// TIA Portal V19 export
FUNCTION "MODE SELECTION" : Void   // FC1, LAD
{ S7_Optimized_Access := 'TRUE' }
// stored: SetENOAutomatically false
   VAR_TEMP   // added for the SCL form of the ladder/FBD networks
      _w1 : Bool;
   END_VAR
BEGIN

REGION Network 1: STANDBY///////////////////////////////////// MGF ////////////////////////////////////////
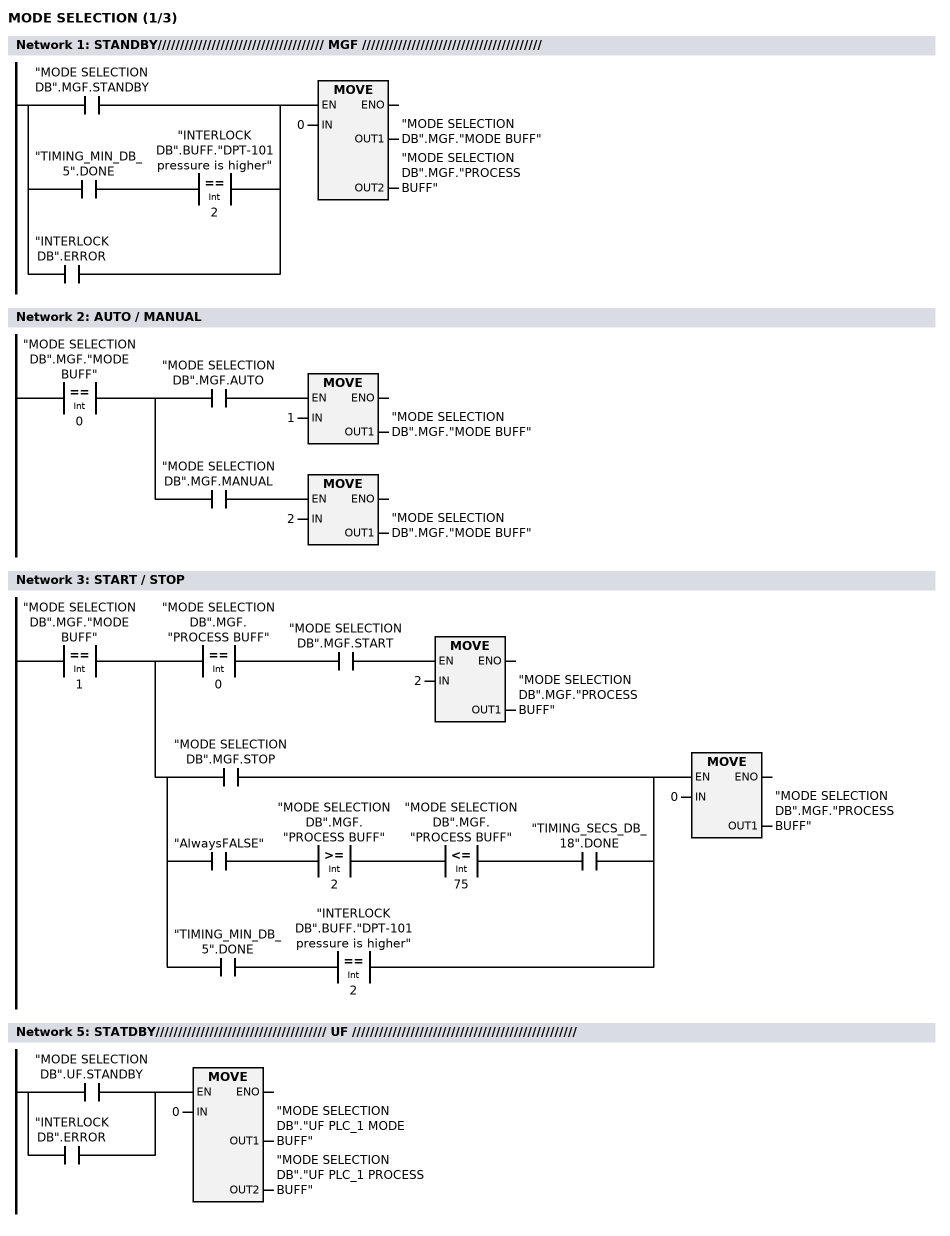
   RUNG wire#powerrail
      Contact( "MODE SELECTION DB".MGF.STANDBY )
      wire#w1
      Move(in := 0, out1 => "MODE SELECTION DB".MGF."MODE BUFF", out2 => "MODE SELECTION DB".MGF."PROCESS BUFF")
   END_RUNG
   RUNG wire#powerrail
      Contact( "TIMING_MIN_DB_5".DONE )
      { S7_Templates := "SrcType := Int" } EQ_Contact(in1 := "INTERLOCK DB".BUFF."DPT-101 pressure is higher", in2 := 2)
   END_RUNG wire#w1
   RUNG wire#powerrail
      Contact( "INTERLOCK DB".ERROR )
   END_RUNG wire#w1
   // the same network as SCL:
   IF "MODE SELECTION DB".MGF.STANDBY OR ("TIMING_MIN_DB_5".DONE AND ("INTERLOCK DB".BUFF."DPT-101 pressure is higher" = 2)) OR "INTERLOCK DB".ERROR THEN
       "MODE SELECTION DB".MGF."MODE BUFF" := 0;
       "MODE SELECTION DB".MGF."PROCESS BUFF" := 0;
   END_IF;
END_REGION

REGION Network 2: AUTO / MANUAL
   RUNG wire#powerrail
      { S7_Templates := "SrcType := Int" } EQ_Contact(in1 := "MODE SELECTION DB".MGF."MODE BUFF", in2 := 0)
      wire#w1
      Contact( "MODE SELECTION DB".MGF.AUTO )
      Move(in := 1, out1 => "MODE SELECTION DB".MGF."MODE BUFF")
   END_RUNG
   RUNG wire#w1
      Contact( "MODE SELECTION DB".MGF.MANUAL )
      Move(in := 2, out1 => "MODE SELECTION DB".MGF."MODE BUFF")
   END_RUNG
   // the same network as SCL:
   #_w1 := "MODE SELECTION DB".MGF."MODE BUFF" = 0;
   IF #_w1 AND "MODE SELECTION DB".MGF.AUTO THEN "MODE SELECTION DB".MGF."MODE BUFF" := 1; END_IF;
   IF #_w1 AND "MODE SELECTION DB".MGF.MANUAL THEN "MODE SELECTION DB".MGF."MODE BUFF" := 2; END_IF;
END_REGION

REGION Network 3: START / STOP
   RUNG wire#powerrail
      { S7_Templates := "SrcType := Int" } EQ_Contact(in1 := "MODE SELECTION DB".MGF."MODE BUFF", in2 := 1)
      wire#w1
      { S7_Templates := "SrcType := Int" } EQ_Contact(in1 := "MODE SELECTION DB".MGF."PROCESS BUFF", in2 := 0)
      Contact( "MODE SELECTION DB".MGF.START )
      Move(in := 2, out1 => "MODE SELECTION DB".MGF."PROCESS BUFF")
   END_RUNG
   RUNG wire#w1
      Contact( "MODE SELECTION DB".MGF.STOP )
      wire#w2
      Move(in := 0, out1 => "MODE SELECTION DB".MGF."PROCESS BUFF")
   END_RUNG
   RUNG wire#w1
      Contact( "AlwaysFALSE" )
      { S7_Templates := "SrcType := Int" } GE_Contact(in1 := "MODE SELECTION DB".MGF."PROCESS BUFF", in2 := 2)
      { S7_Templates := "SrcType := Int" } LE_Contact(in1 := "MODE SELECTION DB".MGF."PROCESS BUFF", in2 := 75)
      Contact( "TIMING_SECS_DB_18".DONE )
   END_RUNG wire#w2
   RUNG wire#w1
      Contact( "TIMING_MIN_DB_5".DONE )
      { S7_Templates := "SrcType := Int" } EQ_Contact(in1 := "INTERLOCK DB".BUFF."DPT-101 pressure is higher", in2 := 2)
   END_RUNG wire#w2
   // the same network as SCL:
   #_w1 := "MODE SELECTION DB".MGF."MODE BUFF" = 1;
   IF #_w1 AND ("MODE SELECTION DB".MGF."PROCESS BUFF" = 0) AND "MODE SELECTION DB".MGF.START THEN
       "MODE SELECTION DB".MGF."PROCESS BUFF" := 2;
   END_IF;
   IF #_w1 AND ("MODE SELECTION DB".MGF.STOP OR ("AlwaysFALSE" AND ("MODE SELECTION DB".MGF."PROCESS BUFF" >= 2) AND ("MODE SELECTION DB".MGF."PROCESS BUFF" <= 75) AND "TIMING_SECS_DB_18".DONE) OR ("TIMING_MIN_DB_5".DONE AND ("INTERLOCK DB".BUFF."DPT-101 pressure is higher" = 2))) THEN
       "MODE SELECTION DB".MGF."PROCESS BUFF" := 0;
   END_IF;
END_REGION

REGION Network 5: STATDBY////////////////////////////////////// UF //////////////////////////////////////////////////
   RUNG wire#powerrail
      Contact( "MODE SELECTION DB".UF.STANDBY )
      wire#w1
      Move(in := 0, out1 => "MODE SELECTION DB"."UF PLC_1 MODE BUFF", out2 => "MODE SELECTION DB"."UF PLC_1 PROCESS BUFF")
   END_RUNG
   RUNG wire#powerrail
      Contact( "INTERLOCK DB".ERROR )
   END_RUNG wire#w1
   // the same network as SCL:
   IF "MODE SELECTION DB".UF.STANDBY OR "INTERLOCK DB".ERROR THEN
       "MODE SELECTION DB"."UF PLC_1 MODE BUFF" := 0;
       "MODE SELECTION DB"."UF PLC_1 PROCESS BUFF" := 0;
   END_IF;
END_REGION

REGION Network 6: AUTO / MANUAL
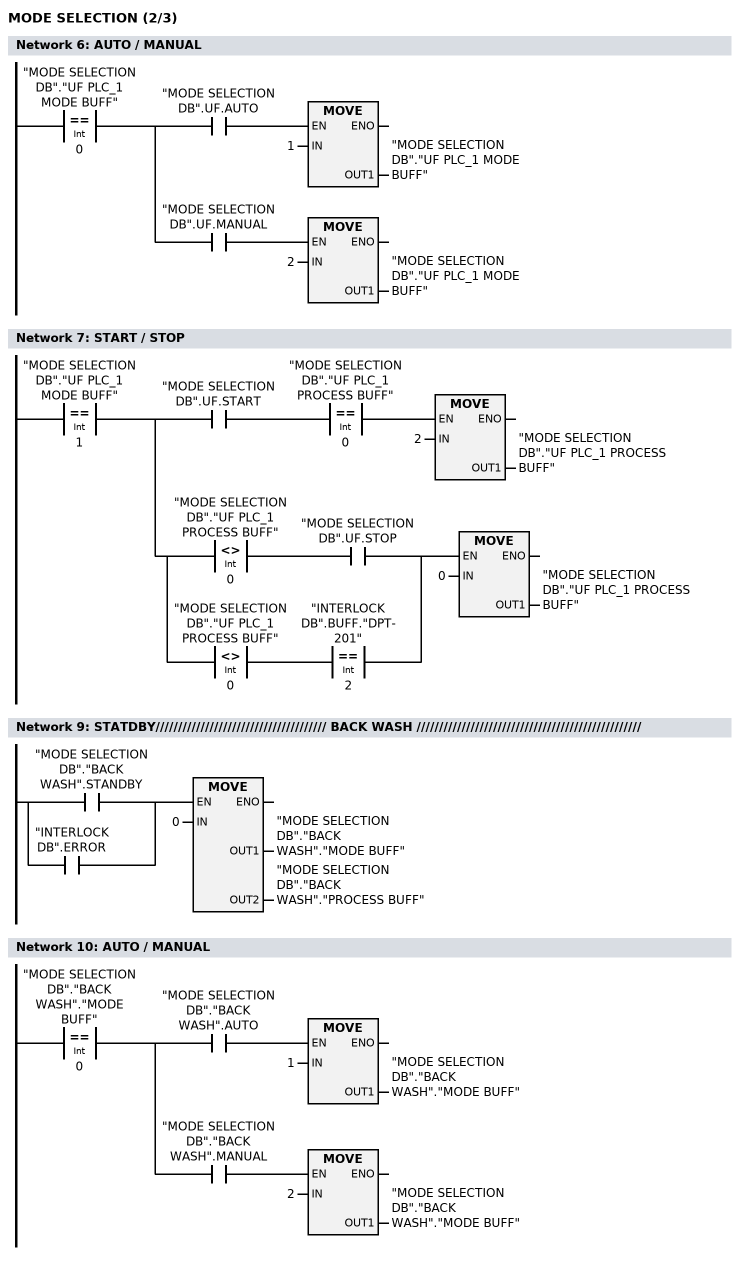
   RUNG wire#powerrail
      { S7_Templates := "SrcType := Int" } EQ_Contact(in1 := "MODE SELECTION DB"."UF PLC_1 MODE BUFF", in2 := 0)
      wire#w1
      Contact( "MODE SELECTION DB".UF.AUTO )
      Move(in := 1, out1 => "MODE SELECTION DB"."UF PLC_1 MODE BUFF")
   END_RUNG
   RUNG wire#w1
      Contact( "MODE SELECTION DB".UF.MANUAL )
      Move(in := 2, out1 => "MODE SELECTION DB"."UF PLC_1 MODE BUFF")
   END_RUNG
   // the same network as SCL:
   #_w1 := "MODE SELECTION DB"."UF PLC_1 MODE BUFF" = 0;
   IF #_w1 AND "MODE SELECTION DB".UF.AUTO THEN "MODE SELECTION DB"."UF PLC_1 MODE BUFF" := 1; END_IF;
   IF #_w1 AND "MODE SELECTION DB".UF.MANUAL THEN "MODE SELECTION DB"."UF PLC_1 MODE BUFF" := 2; END_IF;
END_REGION

REGION Network 7: START / STOP
   RUNG wire#powerrail
      { S7_Templates := "SrcType := Int" } EQ_Contact(in1 := "MODE SELECTION DB"."UF PLC_1 MODE BUFF", in2 := 1)
      wire#w1
      Contact( "MODE SELECTION DB".UF.START )
      { S7_Templates := "SrcType := Int" } EQ_Contact(in1 := "MODE SELECTION DB"."UF PLC_1 PROCESS BUFF", in2 := 0)
      Move(in := 2, out1 => "MODE SELECTION DB"."UF PLC_1 PROCESS BUFF")
   END_RUNG
   RUNG wire#w1
      { S7_Templates := "SrcType := Int" } NE_Contact(in1 := "MODE SELECTION DB"."UF PLC_1 PROCESS BUFF", in2 := 0)
      Contact( "MODE SELECTION DB".UF.STOP )
      wire#w2
      Move(in := 0, out1 => "MODE SELECTION DB"."UF PLC_1 PROCESS BUFF")
   END_RUNG
   RUNG wire#w1
      { S7_Templates := "SrcType := Int" } NE_Contact(in1 := "MODE SELECTION DB"."UF PLC_1 PROCESS BUFF", in2 := 0)
      { S7_Templates := "SrcType := Int" } EQ_Contact(in1 := "INTERLOCK DB".BUFF."DPT-201", in2 := 2)
   END_RUNG wire#w2
   // the same network as SCL:
   #_w1 := "MODE SELECTION DB"."UF PLC_1 MODE BUFF" = 1;
   IF #_w1 AND "MODE SELECTION DB".UF.START AND ("MODE SELECTION DB"."UF PLC_1 PROCESS BUFF" = 0) THEN
       "MODE SELECTION DB"."UF PLC_1 PROCESS BUFF" := 2;
   END_IF;
   IF #_w1 AND ((("MODE SELECTION DB"."UF PLC_1 PROCESS BUFF" <> 0) AND "MODE SELECTION DB".UF.STOP) OR (("MODE SELECTION DB"."UF PLC_1 PROCESS BUFF" <> 0) AND ("INTERLOCK DB".BUFF."DPT-201" = 2))) THEN
       "MODE SELECTION DB"."UF PLC_1 PROCESS BUFF" := 0;
   END_IF;
END_REGION

REGION Network 9: STATDBY////////////////////////////////////// BACK WASH //////////////////////////////////////////////////
   RUNG wire#powerrail
      Contact( "MODE SELECTION DB"."BACK WASH".STANDBY )
      wire#w1
      Move(in := 0, out1 => "MODE SELECTION DB"."BACK WASH"."MODE BUFF", out2 => "MODE SELECTION DB"."BACK WASH"."PROCESS BUFF")
   END_RUNG
   RUNG wire#powerrail
      Contact( "INTERLOCK DB".ERROR )
   END_RUNG wire#w1
   // the same network as SCL:
   IF "MODE SELECTION DB"."BACK WASH".STANDBY OR "INTERLOCK DB".ERROR THEN
       "MODE SELECTION DB"."BACK WASH"."MODE BUFF" := 0;
       "MODE SELECTION DB"."BACK WASH"."PROCESS BUFF" := 0;
   END_IF;
END_REGION

REGION Network 10: AUTO / MANUAL
   RUNG wire#powerrail
      { S7_Templates := "SrcType := Int" } EQ_Contact(in1 := "MODE SELECTION DB"."BACK WASH"."MODE BUFF", in2 := 0)
      wire#w1
      Contact( "MODE SELECTION DB"."BACK WASH".AUTO )
      Move(in := 1, out1 => "MODE SELECTION DB"."BACK WASH"."MODE BUFF")
   END_RUNG
   RUNG wire#w1
      Contact( "MODE SELECTION DB"."BACK WASH".MANUAL )
      Move(in := 2, out1 => "MODE SELECTION DB"."BACK WASH"."MODE BUFF")
   END_RUNG
   // the same network as SCL:
   #_w1 := "MODE SELECTION DB"."BACK WASH"."MODE BUFF" = 0;
   IF #_w1 AND "MODE SELECTION DB"."BACK WASH".AUTO THEN
       "MODE SELECTION DB"."BACK WASH"."MODE BUFF" := 1;
   END_IF;
   IF #_w1 AND "MODE SELECTION DB"."BACK WASH".MANUAL THEN
       "MODE SELECTION DB"."BACK WASH"."MODE BUFF" := 2;
   END_IF;
END_REGION

REGION Network 11: START / STOP
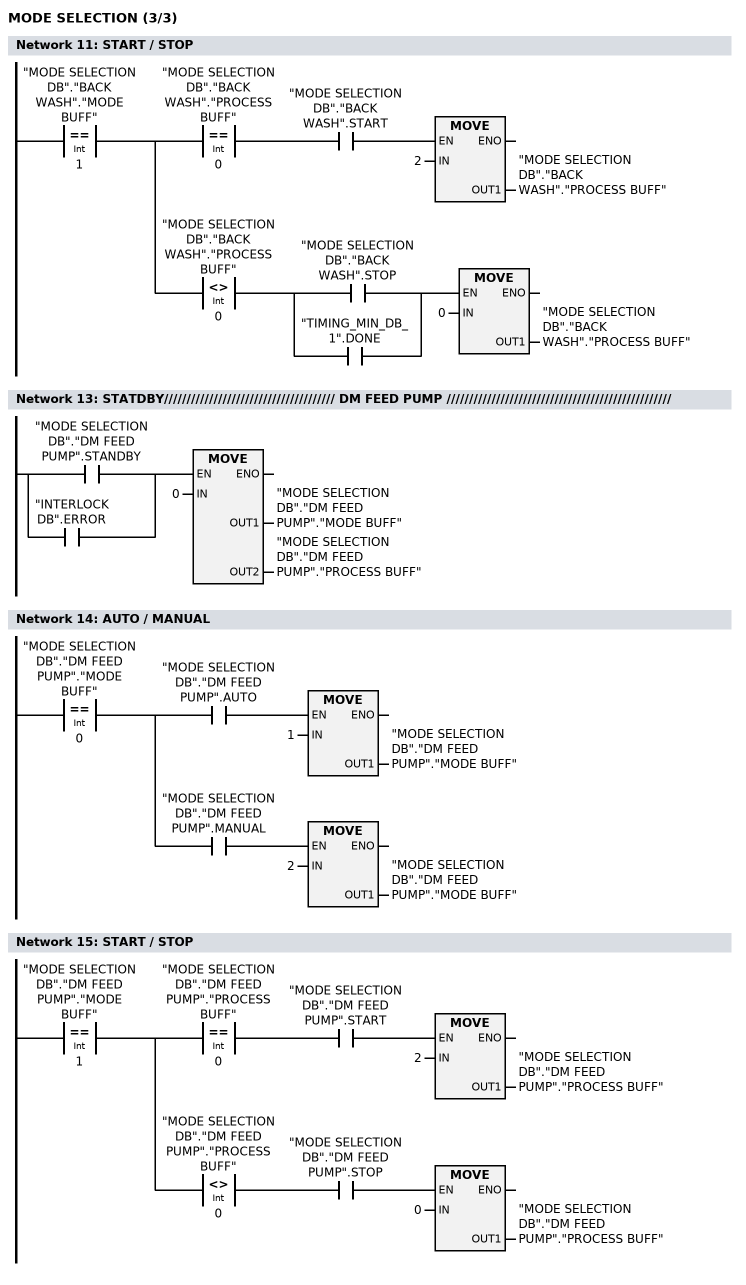
   RUNG wire#powerrail
      { S7_Templates := "SrcType := Int" } EQ_Contact(in1 := "MODE SELECTION DB"."BACK WASH"."MODE BUFF", in2 := 1)
      wire#w1
      { S7_Templates := "SrcType := Int" } EQ_Contact(in1 := "MODE SELECTION DB"."BACK WASH"."PROCESS BUFF", in2 := 0)
      Contact( "MODE SELECTION DB"."BACK WASH".START )
      Move(in := 2, out1 => "MODE SELECTION DB"."BACK WASH"."PROCESS BUFF")
   END_RUNG
   RUNG wire#w1
      { S7_Templates := "SrcType := Int" } NE_Contact(in1 := "MODE SELECTION DB"."BACK WASH"."PROCESS BUFF", in2 := 0)
      wire#w2
      Contact( "MODE SELECTION DB"."BACK WASH".STOP )
      wire#w3
      Move(in := 0, out1 => "MODE SELECTION DB"."BACK WASH"."PROCESS BUFF")
   END_RUNG
   RUNG wire#w2
      Contact( "TIMING_MIN_DB_1".DONE )
   END_RUNG wire#w3
   // the same network as SCL:
   #_w1 := "MODE SELECTION DB"."BACK WASH"."MODE BUFF" = 1;
   IF #_w1 AND ("MODE SELECTION DB"."BACK WASH"."PROCESS BUFF" = 0) AND "MODE SELECTION DB"."BACK WASH".START THEN
       "MODE SELECTION DB"."BACK WASH"."PROCESS BUFF" := 2;
   END_IF;
   IF #_w1 AND ("MODE SELECTION DB"."BACK WASH"."PROCESS BUFF" <> 0) AND ("MODE SELECTION DB"."BACK WASH".STOP OR "TIMING_MIN_DB_1".DONE) THEN
       "MODE SELECTION DB"."BACK WASH"."PROCESS BUFF" := 0;
   END_IF;
END_REGION

REGION Network 13: STATDBY////////////////////////////////////// DM FEED PUMP //////////////////////////////////////////////////
   RUNG wire#powerrail
      Contact( "MODE SELECTION DB"."DM FEED PUMP".STANDBY )
      wire#w1
      Move(in := 0, out1 => "MODE SELECTION DB"."DM FEED PUMP"."MODE BUFF", out2 => "MODE SELECTION DB"."DM FEED PUMP"."PROCESS BUFF")
   END_RUNG
   RUNG wire#powerrail
      Contact( "INTERLOCK DB".ERROR )
   END_RUNG wire#w1
   // the same network as SCL:
   IF "MODE SELECTION DB"."DM FEED PUMP".STANDBY OR "INTERLOCK DB".ERROR THEN
       "MODE SELECTION DB"."DM FEED PUMP"."MODE BUFF" := 0;
       "MODE SELECTION DB"."DM FEED PUMP"."PROCESS BUFF" := 0;
   END_IF;
END_REGION

REGION Network 14: AUTO / MANUAL
   RUNG wire#powerrail
      { S7_Templates := "SrcType := Int" } EQ_Contact(in1 := "MODE SELECTION DB"."DM FEED PUMP"."MODE BUFF", in2 := 0)
      wire#w1
      Contact( "MODE SELECTION DB"."DM FEED PUMP".AUTO )
      Move(in := 1, out1 => "MODE SELECTION DB"."DM FEED PUMP"."MODE BUFF")
   END_RUNG
   RUNG wire#w1
      Contact( "MODE SELECTION DB"."DM FEED PUMP".MANUAL )
      Move(in := 2, out1 => "MODE SELECTION DB"."DM FEED PUMP"."MODE BUFF")
   END_RUNG
   // the same network as SCL:
   #_w1 := "MODE SELECTION DB"."DM FEED PUMP"."MODE BUFF" = 0;
   IF #_w1 AND "MODE SELECTION DB"."DM FEED PUMP".AUTO THEN
       "MODE SELECTION DB"."DM FEED PUMP"."MODE BUFF" := 1;
   END_IF;
   IF #_w1 AND "MODE SELECTION DB"."DM FEED PUMP".MANUAL THEN
       "MODE SELECTION DB"."DM FEED PUMP"."MODE BUFF" := 2;
   END_IF;
END_REGION

REGION Network 15: START / STOP
   RUNG wire#powerrail
      { S7_Templates := "SrcType := Int" } EQ_Contact(in1 := "MODE SELECTION DB"."DM FEED PUMP"."MODE BUFF", in2 := 1)
      wire#w1
      { S7_Templates := "SrcType := Int" } EQ_Contact(in1 := "MODE SELECTION DB"."DM FEED PUMP"."PROCESS BUFF", in2 := 0)
      Contact( "MODE SELECTION DB"."DM FEED PUMP".START )
      Move(in := 2, out1 => "MODE SELECTION DB"."DM FEED PUMP"."PROCESS BUFF")
   END_RUNG
   RUNG wire#w1
      { S7_Templates := "SrcType := Int" } NE_Contact(in1 := "MODE SELECTION DB"."DM FEED PUMP"."PROCESS BUFF", in2 := 0)
      Contact( "MODE SELECTION DB"."DM FEED PUMP".STOP )
      Move(in := 0, out1 => "MODE SELECTION DB"."DM FEED PUMP"."PROCESS BUFF")
   END_RUNG
   // the same network as SCL:
   #_w1 := "MODE SELECTION DB"."DM FEED PUMP"."MODE BUFF" = 1;
   IF #_w1 AND ("MODE SELECTION DB"."DM FEED PUMP"."PROCESS BUFF" = 0) AND "MODE SELECTION DB"."DM FEED PUMP".START THEN
       "MODE SELECTION DB"."DM FEED PUMP"."PROCESS BUFF" := 2;
   END_IF;
   IF #_w1 AND ("MODE SELECTION DB"."DM FEED PUMP"."PROCESS BUFF" <> 0) AND "MODE SELECTION DB"."DM FEED PUMP".STOP THEN
       "MODE SELECTION DB"."DM FEED PUMP"."PROCESS BUFF" := 0;
   END_IF;
END_REGION
END_FUNCTION
